SUBAPPLICATION ACTION_SERVER
  (* Standard: 61499-2 *)
  (* Version 1.0, 2023-04-02, Tim Hesse *)
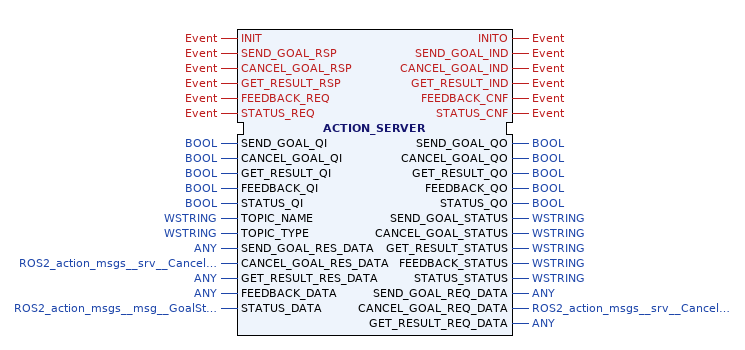
  EVENT_INPUT
    INIT; (* Initialization Request *)
    SEND_GOAL_RSP; (* Normal Execution Request *)
    CANCEL_GOAL_RSP;
    GET_RESULT_RSP;
    FEEDBACK_REQ;
    STATUS_REQ;
  END_EVENT
  EVENT_OUTPUT
    INITO; (* Initialization Confirm *)
    SEND_GOAL_IND; (* Execution Confirmation *)
    CANCEL_GOAL_IND;
    GET_RESULT_IND;
    FEEDBACK_CNF;
    STATUS_CNF;
  END_EVENT
  VAR_INPUT
    SEND_GOAL_QI : BOOL; (* Input event qualifier *)
    CANCEL_GOAL_QI : BOOL;
    GET_RESULT_QI : BOOL;
    FEEDBACK_QI : BOOL;
    STATUS_QI : BOOL;
    TOPIC_NAME : WSTRING;
    TOPIC_TYPE : WSTRING;
    SEND_GOAL_RES_DATA : ANY;
    CANCEL_GOAL_RES_DATA : ROS2_action_msgs__srv__CancelGoal__Response;
    GET_RESULT_RES_DATA : ANY;
    FEEDBACK_DATA : ANY;
    STATUS_DATA : ROS2_action_msgs__msg__GoalStatusArray;
  END_VAR
  VAR_OUTPUT
    SEND_GOAL_QO : BOOL; (* Output event qualifier *)
    CANCEL_GOAL_QO : BOOL;
    GET_RESULT_QO : BOOL;
    FEEDBACK_QO : BOOL;
    STATUS_QO : BOOL;
    SEND_GOAL_STATUS : WSTRING;
    CANCEL_GOAL_STATUS : WSTRING;
    GET_RESULT_STATUS : WSTRING;
    FEEDBACK_STATUS : WSTRING;
    STATUS_STATUS : WSTRING;
    SEND_GOAL_REQ_DATA : ANY;
    CANCEL_GOAL_REQ_DATA : ROS2_action_msgs__srv__CancelGoal__Request;
    GET_RESULT_REQ_DATA : ANY;
  END_VAR
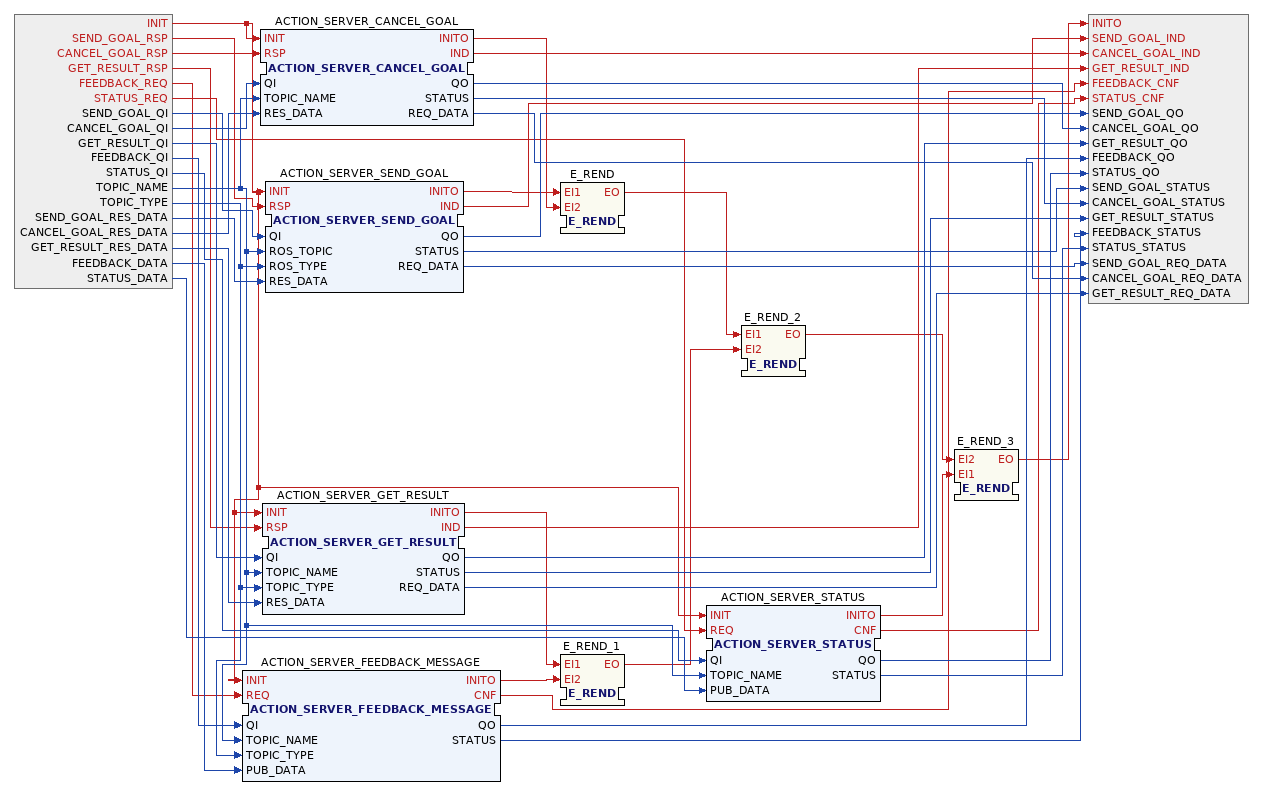
  FBS
    E_REND : E_REND;
    E_REND_1 : E_REND;
    E_REND_2 : E_REND;
    E_REND_3 : E_REND;
  END_FBS
  SUBAPPS
    ACTION_SERVER_SEND_GOAL : ACTION_SERVER_SEND_GOAL;
    ACTION_SERVER_CANCEL_GOAL : ACTION_SERVER_CANCEL_GOAL;
    ACTION_SERVER_GET_RESULT : ACTION_SERVER_GET_RESULT;
    ACTION_SERVER_FEEDBACK_MESSAGE : ACTION_SERVER_FEEDBACK_MESSAGE;
    ACTION_SERVER_STATUS : ACTION_SERVER_STATUS;
  END_SUBAPPS
  EVENT_CONNECTIONS
    E_REND.EO TO E_REND_2.EI1;
    E_REND_1.EO TO E_REND_2.EI2;
    ACTION_SERVER_SEND_GOAL.INITO TO E_REND.EI1;
    ACTION_SERVER_CANCEL_GOAL.INITO TO E_REND.EI2;
    ACTION_SERVER_GET_RESULT.INITO TO E_REND_1.EI1;
    ACTION_SERVER_FEEDBACK_MESSAGE.INITO TO E_REND_1.EI2;
    INIT TO ACTION_SERVER_SEND_GOAL.INIT;
    INIT TO ACTION_SERVER_CANCEL_GOAL.INIT;
    INIT TO ACTION_SERVER_GET_RESULT.INIT;
    INIT TO ACTION_SERVER_FEEDBACK_MESSAGE.INIT;
    SEND_GOAL_RSP TO ACTION_SERVER_SEND_GOAL.RSP;
    CANCEL_GOAL_RSP TO ACTION_SERVER_CANCEL_GOAL.RSP;
    GET_RESULT_RSP TO ACTION_SERVER_GET_RESULT.RSP;
    FEEDBACK_REQ TO ACTION_SERVER_FEEDBACK_MESSAGE.REQ;
    ACTION_SERVER_SEND_GOAL.IND TO SEND_GOAL_IND;
    ACTION_SERVER_CANCEL_GOAL.IND TO CANCEL_GOAL_IND;
    ACTION_SERVER_GET_RESULT.IND TO GET_RESULT_IND;
    ACTION_SERVER_FEEDBACK_MESSAGE.CNF TO FEEDBACK_CNF;
    E_REND_2.EO TO E_REND_3.EI2;
    E_REND_3.EO TO INITO;
    ACTION_SERVER_STATUS.INITO TO E_REND_3.EI1;
    ACTION_SERVER_STATUS.CNF TO STATUS_CNF;
    INIT TO ACTION_SERVER_STATUS.INIT;
    STATUS_REQ TO ACTION_SERVER_STATUS.REQ;
  END_CONNECTIONS
  DATA_CONNECTIONS
    SEND_GOAL_QI TO ACTION_SERVER_SEND_GOAL.QI;
    CANCEL_GOAL_QI TO ACTION_SERVER_CANCEL_GOAL.QI;
    GET_RESULT_QI TO ACTION_SERVER_GET_RESULT.QI;
    FEEDBACK_QI TO ACTION_SERVER_FEEDBACK_MESSAGE.QI;
    TOPIC_NAME TO ACTION_SERVER_SEND_GOAL.ROS_TOPIC;
    TOPIC_NAME TO ACTION_SERVER_CANCEL_GOAL.TOPIC_NAME;
    TOPIC_NAME TO ACTION_SERVER_GET_RESULT.TOPIC_NAME;
    TOPIC_NAME TO ACTION_SERVER_FEEDBACK_MESSAGE.TOPIC_NAME;
    TOPIC_TYPE TO ACTION_SERVER_SEND_GOAL.ROS_TYPE;
    TOPIC_TYPE TO ACTION_SERVER_GET_RESULT.TOPIC_TYPE;
    TOPIC_TYPE TO ACTION_SERVER_FEEDBACK_MESSAGE.TOPIC_TYPE;
    SEND_GOAL_RES_DATA TO ACTION_SERVER_SEND_GOAL.RES_DATA;
    CANCEL_GOAL_RES_DATA TO ACTION_SERVER_CANCEL_GOAL.RES_DATA;
    GET_RESULT_RES_DATA TO ACTION_SERVER_GET_RESULT.RES_DATA;
    FEEDBACK_DATA TO ACTION_SERVER_FEEDBACK_MESSAGE.PUB_DATA;
    ACTION_SERVER_SEND_GOAL.QO TO SEND_GOAL_QO;
    ACTION_SERVER_SEND_GOAL.STATUS TO SEND_GOAL_STATUS;
    ACTION_SERVER_SEND_GOAL.REQ_DATA TO SEND_GOAL_REQ_DATA;
    ACTION_SERVER_CANCEL_GOAL.QO TO CANCEL_GOAL_QO;
    ACTION_SERVER_CANCEL_GOAL.STATUS TO CANCEL_GOAL_STATUS;
    ACTION_SERVER_CANCEL_GOAL.REQ_DATA TO CANCEL_GOAL_REQ_DATA;
    ACTION_SERVER_GET_RESULT.QO TO GET_RESULT_QO;
    ACTION_SERVER_GET_RESULT.STATUS TO GET_RESULT_STATUS;
    ACTION_SERVER_GET_RESULT.REQ_DATA TO GET_RESULT_REQ_DATA;
    ACTION_SERVER_FEEDBACK_MESSAGE.QO TO FEEDBACK_QO;
    ACTION_SERVER_FEEDBACK_MESSAGE.STATUS TO FEEDBACK_STATUS;
    ACTION_SERVER_STATUS.QO TO STATUS_QO;
    ACTION_SERVER_STATUS.STATUS TO STATUS_STATUS;
    STATUS_QI TO ACTION_SERVER_STATUS.QI;
    TOPIC_NAME TO ACTION_SERVER_STATUS.TOPIC_NAME;
    STATUS_DATA TO ACTION_SERVER_STATUS.PUB_DATA;
  END_CONNECTIONS
END_SUBAPPLICATION
